Yaskawa INFORM job: ARUBA_1.JBI

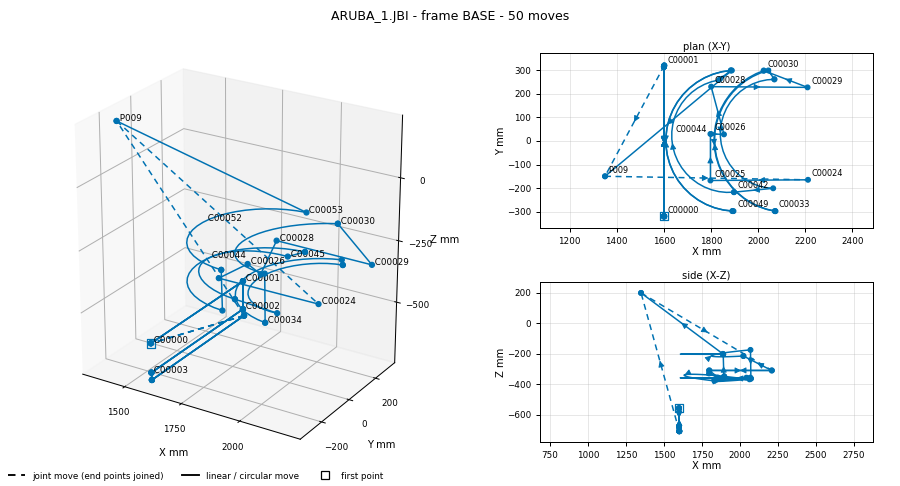
[picture p0: tool path of ARUBA_1.JBI in frame BASE, 50 of 56 moves have a stored position in this frame; points joined in program order, loops and branches not executed]
/JOB
//NAME ARUBA_1
//POS
///NPOS 54,0,54,1,0,2
///TOOL 0
///POSTYPE BASE
///RECTAN
///RCONF 0,0,0,0,0,0,0,0,0,0,0,0,0,0,0,0,0,0,0,0,0,0,0,0
C00000=1600.010,-320.001,-559.985,114.2781,-89.9960,66.7194
C00001=1599.973,314.437,-559.938,-30.8559,-89.9841,-150.1432
C00002=1599.938,314.383,-679.915,-57.7628,-89.9776,-123.2379
C00003=1599.931,-319.990,-679.928,-62.9212,-89.9727,-117.0786
C00004=1601.398,-319.931,-709.869,-179.9782,-50.0144,-0.0232
C00005=1601.406,320.007,-709.860,-179.9770,-50.0151,-0.0241
C00006=1600.010,-320.001,-559.985,114.2781,-89.9960,66.7194
C00007=1599.973,314.437,-559.938,-30.8559,-89.9841,-150.1432
C00008=1599.938,314.383,-679.915,-57.7628,-89.9776,-123.2379
C00009=1599.931,-319.990,-679.928,-62.9212,-89.9727,-117.0786
C00010=1601.398,-319.931,-709.869,-179.9782,-50.0144,-0.0232
C00011=1601.406,320.007,-709.860,-179.9770,-50.0151,-0.0241
C00012=1600.010,-320.001,-559.985,114.2781,-89.9960,66.7194
C00013=1599.973,314.437,-559.938,-30.8559,-89.9841,-150.1432
C00014=1599.938,314.383,-679.915,-57.7628,-89.9776,-123.2379
C00015=1599.931,-319.990,-679.928,-62.9212,-89.9727,-117.0786
C00016=1601.398,-319.931,-709.869,-179.9782,-50.0144,-0.0232
C00017=1601.406,320.007,-709.860,-179.9770,-50.0151,-0.0241
C00018=1600.010,-320.001,-559.985,114.2781,-89.9960,66.7194
C00019=1599.973,314.437,-559.938,-30.8559,-89.9841,-150.1432
C00020=1599.938,314.383,-679.915,-57.7628,-89.9776,-123.2379
C00021=1599.931,-319.990,-679.928,-62.9212,-89.9727,-117.0786
C00022=1601.398,-319.931,-709.869,-179.9782,-50.0144,-0.0232
C00023=1601.406,320.007,-709.860,-179.9770,-50.0151,-0.0241
///RCONF 0,0,0,0,1,0,0,0,0,0,0,0,0,0,0,0,0,0,0,0,0,0,0,0
C00024=2211.411,-164.885,-310.009,-178.8281,-29.9756,87.6555
C00025=1797.383,-167.804,-309.883,-179.9751,-29.9966,89.9599
C00026=1797.336,29.624,-329.788,-179.9887,-0.0046,89.9431
///RCONF 1,0,0,0,0,0,0,0,0,0,0,0,0,0,0,0,0,0,0,0,0,0,0,0
C00027=1854.817,27.910,-356.495,138.1150,0.4795,88.8071
///RCONF 0,0,0,0,0,0,0,0,0,0,0,0,0,0,0,0,0,0,0,0,0,0,0,0
C00028=1800.515,230.389,-310.328,-178.5752,-29.3550,-91.9736
C00029=2209.491,227.290,-310.238,-179.1455,-29.3776,-90.8166
C00030=2023.524,298.371,-215.002,-155.5081,-88.2298,-114.0488
C00031=2023.524,298.371,-215.002,-155.5081,-88.2298,-114.0488
C00032=1813.423,26.953,-215.002,-156.9343,-88.2466,-22.6259
///RCONF 0,0,0,1,0,0,0,0,0,0,0,0,0,0,0,0,0,0,0,0,0,0,0,0
C00033=2070.189,-297.808,-174.781,167.5563,-88.3453,103.8852
C00034=2072.884,-297.904,-363.667,-158.2647,-88.2591,69.6900
C00035=2072.884,-297.904,-363.667,-158.2647,-88.2591,69.6900
///RCONF 0,0,0,0,0,0,0,0,0,0,0,0,0,0,0,0,0,0,0,0,0,0,0,0
C00036=1815.735,25.568,-362.142,-158.2790,-88.2777,-21.2521
C00037=2043.124,299.197,-357.550,172.0781,-88.3860,-82.6051
C00038=2068.758,261.489,-358.008,-177.9538,-56.3805,-93.0897
C00039=2068.758,261.489,-358.008,-177.9538,-56.3805,-93.0897
C00040=1839.205,25.661,-381.923,-177.9546,-56.3859,-1.0844
///RCONF 0,0,0,1,0,0,0,0,0,0,0,0,0,0,0,0,0,0,0,0,0,0,0,0
C00041=2063.699,-200.924,-368.491,-179.4452,-56.4081,91.6963
C00042=1897.190,-217.395,-348.882,-179.4561,-56.4122,91.7088
C00043=1897.190,-217.394,-348.890,-179.4569,-56.4120,91.7090
///RCONF 0,0,0,0,0,0,0,0,0,0,0,0,0,0,0,0,0,0,0,0,0,0,0,0
C00044=1633.002,20.692,-341.256,-177.9115,-56.4043,-2.1191
C00045=1832.992,258.509,-378.743,179.0999,-56.4261,-89.5361
C00046=1884.056,299.188,-363.146,170.7208,-88.4059,-81.2280
C00047=1884.056,299.188,-363.146,170.7208,-88.4059,-81.2280
C00048=1610.189,40.360,-358.670,-154.6250,-88.2603,-24.9017
///RCONF 0,0,0,1,0,0,0,0,0,0,0,0,0,0,0,0,0,0,0,0,0,0,0,0
C00049=1895.222,-297.835,-361.532,-155.2341,-88.2757,66.6826
C00050=1890.715,-297.656,-203.952,-155.1285,-88.2790,66.5874
C00051=1890.715,-297.656,-203.952,-155.1285,-88.2790,66.5874
///RCONF 0,0,0,0,0,0,0,0,0,0,0,0,0,0,0,0,0,0,0,0,0,0,0,0
C00052=1610.132,33.670,-202.330,169.6337,-88.4395,10.8750
C00053=1888.278,299.196,-200.812,171.7400,-88.4493,-82.2282
///POSTYPE PULSE
///PULSE
EC00000=0
EC00001=0
EC00002=0
EC00003=0
EC00004=0
EC00005=0
EC00006=92160
EC00007=92160
EC00008=92160
EC00009=92160
EC00010=92160
EC00011=92160
EC00012=184320
EC00013=184320
EC00014=184320
EC00015=184320
EC00016=184320
EC00017=184320
EC00018=276480
EC00019=276480
EC00020=276480
EC00021=276480
EC00022=276480
EC00023=276480
EC00024=92160
EC00025=92160
EC00026=92160
EC00027=92160
EC00028=92160
EC00029=92160
EC00030=92160
EC00031=92160
EC00032=92160
EC00033=92160
EC00034=92160
EC00035=92160
EC00036=92160
EC00037=92160
EC00038=92160
EC00039=92160
EC00040=92160
EC00041=92160
EC00042=276480
EC00043=276480
EC00044=276480
EC00045=276480
EC00046=276480
EC00047=276480
EC00048=276480
EC00049=276480
EC00050=276480
EC00051=276480
EC00052=276480
EC00053=276480
///POSTYPE BASE
///RECTAN
///RCONF 1,0,0,0,0,0,0,0,0,0,0,0,0,0,0,0,0,0,0,0,0,0,0,0
P00009=1350.000,-150.000,200.000,-180.0000,-45.0000,0.0000
///POSTYPE PULSE
///PULSE
EX00000=0
EX00001=92160
//INST
///DATE 2023/06/22 11:31
///ATTR SC,RW,RJ
////FRAME BASE
///GROUP1 RB1,ST1
NOP
MOVJ C00000 EC00000 VJ=12.00
CALL JOB:SPYON
MOVL C00001 EC00001 V=200.0
MOVL C00002 EC00002 V=200.0
MOVL C00003 EC00003 V=200.0
MOVL C00004 EC00004 V=200.0
MOVL C00005 EC00005 V=200.0
CALL JOB:SPYOF
MOVJ C00006 EC00006 VJ=12.00
CALL JOB:SPYON
MOVL C00007 EC00007 V=200.0
MOVL C00008 EC00008 V=200.0
MOVL C00009 EC00009 V=200.0
MOVL C00010 EC00010 V=200.0
MOVL C00011 EC00011 V=200.0
CALL JOB:SPYOF
MOVJ C00012 EC00012 VJ=12.00
CALL JOB:SPYON
MOVL C00013 EC00013 V=200.0
MOVL C00014 EC00014 V=200.0
MOVL C00015 EC00015 V=200.0
MOVL C00016 EC00016 V=200.0
MOVL C00017 EC00017 V=200.0
CALL JOB:SPYOF
MOVJ C00018 EC00018 VJ=12.00
CALL JOB:SPYON
MOVL C00019 EC00019 V=200.0
MOVL C00020 EC00020 V=200.0
MOVL C00021 EC00021 V=200.0
MOVL C00022 EC00022 V=200.0
MOVL C00023 EC00023 V=200.0
CALL JOB:SPYOF
MOVJ P009 EX001 VJ=12.00
MOVJ C00024 EC00024 VJ=12.00
CALL JOB:SPYON
MOVL C00025 EC00025 V=200.0
MOVL C00026 EC00026 V=200.0
MOVL C00027 EC00027 V=200.0
CALL JOB:SPYOF
MOVL C00028 EC00028 V=200.0
CALL JOB:SPYON
MOVL C00029 EC00029 V=200.0
CALL JOB:SPYOF
MOVL C00030 EC00030 V=200.0
CALL JOB:SPYON
MOVC C00031 EC00031 V=200.0
MOVC C00032 EC00032 V=200.0
MOVC C00033 EC00033 V=200.0
MOVL C00034 EC00034 V=200.0
MOVC C00035 EC00035 V=200.0
MOVC C00036 EC00036 V=200.0
MOVC C00037 EC00037 V=200.0
MOVL C00038 EC00038 V=200.0
MOVC C00039 EC00039 V=200.0
MOVC C00040 EC00040 V=200.0
MOVC C00041 EC00041 V=200.0
CALL JOB:SPYOF
MOVL C00042 EC00042 V=200.0
CALL JOB:SPYON
MOVC C00043 EC00043 V=200.0
MOVC C00044 EC00044 V=200.0
MOVC C00045 EC00045 V=200.0
MOVL C00046 EC00046 V=200.0
MOVC C00047 EC00047 V=200.0
MOVC C00048 EC00048 V=200.0
MOVC C00049 EC00049 V=200.0
MOVL C00050 EC00050 V=200.0
MOVC C00051 EC00051 V=200.0
MOVC C00052 EC00052 V=200.0
MOVC C00053 EC00053 V=200.0
CALL JOB:SPYOF
MOVL P009 EX000 V=200.0
END
